// TwinCAT 3 PLC project PLC
// ProgramVersion: 3.1.4022.3
// libraries:
//   Tc2_EtherCAT, * (Beckhoff Automation GmbH)
//   Tc2_Math, * (Beckhoff Automation GmbH)
//   Tc2_Standard, * (Beckhoff Automation GmbH)
//   Tc2_System, * (Beckhoff Automation GmbH)
//   Tc2_TcpIp, * (Beckhoff Automation GmbH)
//   Tc2_Utilities, * (Beckhoff Automation GmbH)
//   Tc3_JsonXml, * (Beckhoff Automation GmbH)
//   Tc3_Module, * (Beckhoff Automation GmbH)
//   Tc3_System_DK, * (Beckhoff - DK)
// project tree:
//   DAQ/FromLib/Influxdb/Reader/ E_InfluxReaderState.TcDUT, FB_InfluxReader.TcPOU
//   DAQ/FromLib/Influxdb/Sender/ FB_InfluxDataCollector.TcPOU, FB_InfluxDataSender.TcPOU
//   DAQ/FromLib/Influxdb/Utils/ ST_InfluxBuffer.TcDUT
//   DAQ/FromLib/StringBuilder/ FB_StringBuilder.TcPOU
//   DAQ/FromLib/TcpIp Connection/ E_TcpState.TcDUT, FB_TcpConnection.TcPOU
//   DAQ/ InfluxAddData_1000Hz.TcPOU, InfluxAddData_100Hz.TcPOU, InfluxAddData_10Hz.TcPOU, InfluxAddData_1Hz.TcPOU, P_InfluxDatabaseWriter.TcPOU, P_InfluxDataCollector.TcPOU
//   DAQ/InfluxReader/ExtractValuesFromInflux/ fcnExtractInfluxData.TcPOU, ST_NumberInString.TcDUT
//   DAQ/InfluxReader/ FB_Flender_DamageReader.TcPOU, P_FlenderGetDamage.TcPOU
//   / DAQ_Collector.TcTTO, DAQ_Writer.TcTTO, MAIN.TcPOU, PlcTask.TcTTO
//   GVLs/ Communication.TcGVL, PersistentVariables.TcGVL
//   HMI/ ST_FROM_HMI.TcDUT, ST_GUI_HMI.TcDUT, ST_HOUR_COUNTERS.TcDUT, ST_PARAMETERS_HMI.TcDUT, ST_TO_HMI.TcDUT
//   Interfaces/JetsonTx2/ ST_JetsonTx2.TcDUT
//   Interfaces/Sick/ ST_SICK.TcDUT
//   Main/Enumerators/ E_EmulatedState.TcDUT
//   Main/Programs/ P_UpdateDAQ.TcPOU, P_UpdateHmi.TcPOU
//   Main/Structures/GPS/ ST_GPS.TcDUT, ST_GPS_CALCULATIONS.TcDUT, ST_GPS_INPUTS.TcDUT, ST_GPS_OUTPUTS.TcDUT
//   Main/Structures/ ST_DATA.TcDUT, ST_PlcTiming.TcDUT
// real-time tasks:
//   TASK PlcTask: cycle T#1ms, priority 20, ADS port 350
//   TASK DAQ_Collector: cycle T#10ms, priority 3, ADS port 351
//   TASK DAQ_Writer: cycle T#100000us, priority 2, ADS port 352

CONFIGURATION PLC
    RESOURCE PLC ON TwinCAT3
        TASK DAQ_Collector(INTERVAL := T#10ms, PRIORITY := 3);
        TASK DAQ_Writer(INTERVAL := T#100000us, PRIORITY := 2);
        TASK PlcTask(INTERVAL := T#1ms, PRIORITY := 20);
        PROGRAM P_InfluxDataCollector WITH DAQ_Collector : P_InfluxDataCollector;
        PROGRAM P_InfluxDatabaseWriter WITH DAQ_Writer : P_InfluxDatabaseWriter;
        PROGRAM MAIN WITH PlcTask : MAIN;
    END_RESOURCE
END_CONFIGURATION

// ---- DAQ/FromLib/Influxdb/Reader/E_InfluxReaderState.TcDUT
{attribute 'qualified_only'}
{attribute 'strict'}
TYPE E_InfluxReaderState :
(
	Idle := 0,
	Connecting,
	Query,
	ConvertingNumbers, 
	Disconnecting
) DINT;
END_TYPE

// ---- DAQ/FromLib/Influxdb/Utils/ST_InfluxBuffer.TcDUT
TYPE ST_InfluxBuffer :
STRUCT
	Initialized : BOOL;
	ReadyToSend	: BOOL;
	Data 		: FB_STRINGBUILDER; 
END_STRUCT
END_TYPE

// ---- DAQ/FromLib/TcpIp Connection/E_TcpState.TcDUT
{attribute 'qualified_only'}
{attribute 'strict'}
TYPE E_TcpState :
(
	None := 0,
	Disconnecting,
	Disconnected,
	Connecting,	
	Connected,
	Sending,
	SendingByReference,
	Waiting,
	Receiving,
	Received
) DINT;
END_TYPE

// ---- DAQ/InfluxReader/ExtractValuesFromInflux/ST_NumberInString.TcDUT
TYPE ST_NumberInString :
STRUCT
	StartIndex : DINT;
	EndIndex	: DINT; 
	Length		: DINT;
	Txt			: T_MAXSTRING;
	Value		: LREAL; 	
END_STRUCT
END_TYPE

// ---- HMI/ST_FROM_HMI.TcDUT
TYPE ST_FROM_HMI :
STRUCT
END_STRUCT
END_TYPE

// ---- HMI/ST_GUI_HMI.TcDUT
TYPE ST_GUI_HMI :
STRUCT
END_STRUCT
END_TYPE

// ---- HMI/ST_HOUR_COUNTERS.TcDUT
TYPE ST_HOUR_COUNTERS :
STRUCT
	
	TotalHours		: LTIME;
	
	WorkingHours	: LTIME;
END_STRUCT
END_TYPE

// ---- HMI/ST_PARAMETERS_HMI.TcDUT
TYPE ST_PARAMETERS_HMI :
STRUCT
END_STRUCT
END_TYPE

// ---- HMI/ST_TO_HMI.TcDUT
TYPE ST_TO_HMI :
STRUCT
	Data		: ST_DATA;
END_STRUCT
END_TYPE

// ---- Interfaces/JetsonTx2/ST_JetsonTx2.TcDUT
TYPE ST_JetsonTx2 :
STRUCT
END_STRUCT
END_TYPE

// ---- Interfaces/Sick/ST_SICK.TcDUT
TYPE ST_SICK :
STRUCT
END_STRUCT
END_TYPE

// ---- Main/Enumerators/E_EmulatedState.TcDUT
TYPE E_EmulatedState :
(
	StaticData := 0,
	SimulinkPlant,
	VirtualPlant,
	PhysicalPlant	
) DINT;
END_TYPE

// ---- Main/Structures/GPS/ST_GPS.TcDUT
TYPE ST_GPS :
STRUCT
	Inputs			: ST_GPS_INPUTS;
	Outputs			: ST_GPS_OUTPUTS;
	Calculations	: ST_GPS_CALCULATIONS;
END_STRUCT
END_TYPE

// ---- Main/Structures/GPS/ST_GPS_CALCULATIONS.TcDUT
TYPE ST_GPS_CALCULATIONS :
STRUCT
END_STRUCT
END_TYPE

// ---- Main/Structures/GPS/ST_GPS_INPUTS.TcDUT
TYPE ST_GPS_INPUTS :
STRUCT
	x			: LREAL;
END_STRUCT
END_TYPE

// ---- Main/Structures/GPS/ST_GPS_OUTPUTS.TcDUT
TYPE ST_GPS_OUTPUTS :
STRUCT
END_STRUCT
END_TYPE

// ---- Main/Structures/ST_DATA.TcDUT
TYPE ST_DATA :
STRUCT
	Timing				: ST_PlcTiming;
	JetsonTx2			: ST_JetsonTx2;
	Sick				: ST_SICK;
	Gps					: ST_Gps;
END_STRUCT
END_TYPE

// ---- Main/Structures/ST_PlcTiming.TcDUT
TYPE ST_PlcTiming :
STRUCT
	TimeStamp 		: T_FILETIME;  	(* Current Windows timestamp *)
	UnixTimeStamp 	: ULINT; 		(* Number of 100 ns since 1.1.1970 *)
	SpanTime		: LTIME;		(* PLC RunTime*)

	ScanTime		: LTIME; 		(* TIME: PLC Scantime *)
	ScanTime_s		: LREAL; 		(* LREAL: PLC Scantime in seconds *)
	ScanTime_ms		: LREAL	:= ScanTime_s * 1E3;		(* LREAL: PLC Scantime in milli seconds *)
	
	Tick			: UDINT := 0; 	(* Current PLC tick count *)
	Toggle			: BOOL; 		(* BOOL: Toggle Each Scan *)
	Toggle1Hz		: BOOL; 		(* BOOL: Toggle at 1 Hz: 1000 ms *)
	Toggle100Hz		: BOOL; 		(* BOOL: Toggle at 100 Hz: 10 ms*)
END_STRUCT
END_TYPE

// ---- GVLs/Communication.TcGVL
{attribute 'qualified_only'}
VAR_GLOBAL
	ToHmi				: ST_TO_HMI;
	
	FromHmi				: ST_FROM_HMI;
	
	Parameters 			: ST_PARAMETERS_HMI;

	Gui					: ST_GUI_HMI; 
	
	HourCounters		: ST_HOUR_COUNTERS;
	
	// Temp
	MyBoolVariable		: BOOL;
END_VAR

// ---- GVLs/PersistentVariables.TcGVL
{attribute 'qualified_only'}
VAR_GLOBAL
	HourCounters		: ST_HOUR_COUNTERS;
END_VAR

// ---- DAQ/P_InfluxDataCollector.TcPOU
PROGRAM P_InfluxDataCollector
VAR 
	Data : REFERENCE TO ST_DATA := P_UpdateDAQ.DataDaq;  
	Tick : LREAL; 
	ActualBufferTime : TIME; 
	
	InfluxData : FB_InfluxDataCollector; 

	Timer1Hz 	: TON; 
	Timer10Hz 	: TON; 
	Timer100Hz 	: TON; 	

END_VAR

Tick := Tick + 1;
RunTimers(); 

// ========= Initialize Data
	InfluxData.Initialize( 	HostName 		:= 'MachinePLC',			// <<---- 	Change to Descriptive MachinePLC name, eg: MachinePLC_TLU 
							Database 		:= 'RD',			// <<---- 	Change to Database name. Needs to be setup beforehand.
							Measurement 	:= 'CKD_Test');	// <<---- 	Measurentname in database. Eg: LORCHALT
// ========= Add Data tags.
// These are written to each "point" i.e. for each ms.
// Add eg: Current State of TestBench - for easy search later on
															
	//Data.AddTag('State','Default');						

// ========= Add Actual Data

	InfluxData.AddLreal('Tick', Tick);

// ======== 1 Hz Data
	IF Time_1Hz THEN
		InfluxData.AddLreal('Test1Hz', 1);	
	
		InfluxAddData_1Hz(		Data 			:= Data,
								DataCollector 	:=  InfluxData); 	
						
	END_IF
	
// ======== 10 Hz Data
	IF Time_10Hz THEN
		InfluxData.AddLreal('Test10Hz', 10);
	
		InfluxAddData_10Hz(	Data 			:= Data,
								DataCollector 	:=  InfluxData); 		
		
	END_IF

// ======== 100 Hz Data
	IF Time_100Hz THEN
		InfluxData.AddLreal('Test100Hz', 100);
	
		InfluxAddData_100Hz(	Data 			:= Data,
								DataCollector 	:=  InfluxData); 

		InfluxAddData_1000Hz(	Data 			:= Data,
								DataCollector 	:=  InfluxData); 
	
								
	END_IF


// =========== Add TimeStamp and start new "point"
InfluxData.AddTimeStamp(ActualBufferTime => ActualBufferTime); 















ResetTimersIfDone();

METHOD ResetTimersIfDone : BOOL
IF Timer1Hz.Q THEN
	Timer1Hz(IN := FALSE); 
	Timer1Hz(IN := TRUE); 

END_IF
IF Timer10Hz.Q THEN
	Timer10Hz(IN := FALSE); 
	Timer10Hz(IN := TRUE); 
	

END_IF
IF Timer100Hz.Q THEN
	Timer100Hz(IN := FALSE); 
	Timer100Hz(IN := TRUE); 
	
END_IF
END_METHOD

METHOD RunTimers : BOOL
Timer1Hz(	IN := TRUE, PT := T#1S		); 
Timer10Hz(	IN := TRUE, PT := T#100MS	); 
Timer100Hz(	IN := TRUE, PT := T#10MS	);
END_METHOD

PROPERTY Time_100Hz : BOOL
GET
Time_100Hz := Timer100Hz.Q;
END_GET
END_PROPERTY

PROPERTY Time_10Hz : BOOL
GET
Time_10Hz := Timer10Hz.Q;
END_GET
END_PROPERTY

PROPERTY Time_1Hz : BOOL
GET
Time_1Hz := Timer1Hz.Q;
END_GET
END_PROPERTY

END_PROGRAM

// ---- Main/Programs/P_UpdateDAQ.TcPOU
PROGRAM P_UpdateDAQ
VAR_IN_OUT
	Data	: ST_DATA;
END_VAR
VAR
	DataDaq : ST_DATA;
END_VAR

DataDaq := Data;

END_PROGRAM

// ---- DAQ/FromLib/Influxdb/Sender/FB_InfluxDataCollector.TcPOU
FUNCTION_BLOCK FB_InfluxDataCollector
VAR
//Writer
	_NameValuePairs			: UDINT; 
	_PointsAdded			: UDINT; 
	
// Misc
	_fbGetSystemTime		: GetSystemTime;
	_bufferTime				: TIME; 
	_fbTimer				: TON; 
END_VAR
VAR
	BufferInUse		: DINT := 1; 
	Buffer1			: ST_InfluxBuffer;
	Buffer2			: ST_InfluxBuffer;
END_VAR
VAR
	iContentLengthIndex : UDINT; 
	iContentLengthBegin : UDINT;
	iContentLengthEnd	: UDINT;
	iContentLength		: UDINT; 
	strContentLength	: T_MAXSTRING; 
END_VAR

METHOD AddBareString : BOOL
VAR_INPUT
	input : T_MaxString; 
END_VAR
DataString.Append(input);
END_METHOD

METHOD PUBLIC AddBool : BOOL
VAR_INPUT
	Name 	: T_MaxString;
	Value 	: BOOL; 
END_VAR
AddName(Name);
IF Value THEN
	DataString.Append('1');
ELSE
	DataString.Append('0');
END_IF
END_METHOD

METHOD PUBLIC AddData : BOOL
VAR_INPUT
	Name 	: T_MaxString;
	Value 	: T_MaxString; 
END_VAR
AddName(Name);
DataString.Append(Value);


_NameValuePairs := _NameValuePairs + 1;
END_METHOD

METHOD AddLreal : BOOL
VAR_INPUT
	Name 	: T_MaxString;
	Value 	: LREAL; 
END_VAR
VAR_INST
	json	: FB_JsonSaxWriter; 
END_VAR
AddName(Name);

json.ResetDocument(); 
json.AddLreal(Value); 
DataString.Append(json.GetDocument());
END_METHOD

METHOD PRIVATE AddName : BOOL
VAR_INPUT
	Name 	: T_MaxString;
END_VAR
IF _NameValuePairs = 0 THEN
	DataString.Append(' ');
ELSE
	DataString.Append(',');
END_IF
DataString.Append(Name);
DataString.Append('=');

_NameValuePairs := _NameValuePairs + 1;
END_METHOD

METHOD AddTag : BOOL
VAR_INPUT
	Key		: T_MAXSTRING;
	Value	: T_MAXSTRING; 
END_VAR
Datastring.Append(',');
Datastring.Append(Key);
DataString.Append('=');
DataString.Append(Value);
END_METHOD

METHOD AddTimeStamp : BOOL; 

VAR
	b : BOOL; 
	SizeLimit : UDINT := 10000000; //10 MB
END_VAR
VAR_OUTPUT
	ActualBufferTime : TIME; 
END_VAR
VAR_INST
	_actualBufferTime : TIME; 
END_VAR
_PointsAdded := _PointsAdded + 1;

DataString.Append(' ');
DataString.Append(ULINT_TO_STRING(CurrentTimeStamp));
DataString.Append('$N');

_fbTimer(	IN := TRUE,
			PT := _bufferTime);
			
IF _fbTimer.Q OR BufferUsed >= 0.9 OR DataString.Length > SizeLimit THEN
	_actualBufferTime := _fbTimer.ET;

	// ======= Add HTTP Content Length
	
		iContentLengthEnd := DataString.Length; 
		
		// Calcualte ContentLength 
		iContentLength := iContentLengthEnd - iContentLengthBegin; 
		strContentLength := TO_STRING(iContentLength); 
		
		// Add content Length to HTTP Header
		memcpy(DataString.StringPointer + iContentLengthIndex, ADR(strContentLength), LEN(strContentLength));


	SetBufferAsReady();
	SwitchBuffer(); 
	Reset(); 
	SetBufferAsNotReady();
	
	
	
	
END_IF

ActualBufferTime := _actualBufferTime;
END_METHOD

PROPERTY BufferOverflow : BOOL
GET
BufferOverflow := DataString.Length = DataString.BufferSize;
END_GET
END_PROPERTY

PROPERTY BufferUsed : LREAL
GET
BufferUsed := UDINT_TO_LREAL(DataString.Length) / UDINT_TO_LREAL(DataString.BufferSize);
END_GET
END_PROPERTY

PROPERTY PROTECTED CurrentTimeStamp : ULINT;
GET
VAR
	normTime	: T_FILETIME;

	dcTime	: T_DCTIME64; 	

	timeLoDW				: ULINT;
	timeHiDW				: ULINT;
	ulTime					: ULINT;
	unixTimeFileTimeDiff	: ULINT;

	
END_VAR
(****************************************************************************************************************

In TwinCAT we get accure timestamp  via GetSystemTime() function block, but it returns so called "filetime"
	filemtime is count of "100 nanoseconds" since 1.1.1601.
	
InfluxDb uses Unix time stamp with accuracy of 1ns. 
	Unix time stamp is seconds since 1.1.1970. 

1.1.1970 - 1.1.1601 in "100 nanoseconds" is 116444736000000000	
*******************************************************************************************************************)

unixTimeFileTimeDiff := 116444736000000000; 
_fbGetSystemTime();
timeHiDW 	:= _fbGetSystemTime.timeHiDW;
timeLoDW 	:= _fbGetSystemTime.timeLoDW; 


normTime := DCTIME64_TO_FILETIME(F_GETCURDCTASKTIME64()); 

normTime.dwHighDateTime := normTime.dwHighDateTime;
normTime.dwLowDateTime := normTime.dwLowDateTime;


ulTime 	:= timeHiDW * 16#FFFFFFFF + timeLoDW; 	// "100 nanoseconds" since 1.1.1601.

//ulTime 	:= normTime.dwHighDateTime * 16#FFFFFFFF + normTime.dwLowDateTime; 	// "100 nanoseconds" since 1.1.1601.

ulTime 	:= ulTime - unixTimeFileTimeDiff;		// "100 nanoseconds" since 1.1.1970.
CurrentTimeStamp 	:= ulTime * 100;						// nanoseconds since 1.1.1970.
END_GET
END_PROPERTY

PROPERTY DataLength : UDINT
GET
DataLength := DataString.Length;
END_GET
END_PROPERTY

PROPERTY DataString : REFERENCE TO FB_STRINGBUILDER
GET
DataString REF= GetData(BufferInUse);
END_GET
END_PROPERTY

METHOD GetData : REFERENCE TO FB_STRINGBUILDER
VAR_INPUT
	BufferNumber : DINT; 
END_VAR

IF BufferNumber = 1 THEN
	GetData REF= Buffer1.Data;
ELSIF BufferNumber = 2 THEN
	GetDAta REF= Buffer2.Data; 
END_IF
END_METHOD

PROPERTY HttpRequest : T_MAXSTRING
GET
HttpRequest := DataString.ToString;
END_GET
END_PROPERTY

METHOD Initialize : BOOL
VAR_INPUT
	HostName 		: T_MAXSTRING;
	Database 		: T_MAXSTRING;  
	Measurement 	: T_MAXSTRING; 
END_VAR
VAR
	MaxBufferTime : TIME := T#2s; 
END_VAR
IF DataString.Length = 0 THEN
	// ============ Build HTTP Header
	DataString.Append('POST /write?db=');
	DataString.Append(Database);
	DataString.AppendLine(' HTTP/1.1');
	
	DataString.Append('Host: ');
	DataString.AppendLine(HostName);
	DataString.AppendLine('User-Agent: TwinCAT HttpClient');
	DataString.AppendLine('Content-Type: application/x-www-form-urlencoded');
	
	DataString.Append('Content-Length: ');
	iContentLengthIndex := DataString.Length; 
	
	DataString.Append('                    '); // Add 10 spaces for adding ContentLength later;
	DataString.AppendLine('');
	DataString.AppendLine(''); 	// <<--- End of HTTP Header
	
	iContentLengthBegin := DataString.Length; 
END_IF

	
// ========== Add host to influx measurement
SetupCollection(Measurement, HostName, MaxBufferTime);
END_METHOD

METHOD IsReadyToSend : BOOL
VAR_INPUT
	BufferNumber : DINT; 
END_VAR
IF BufferNumber = 1 THEN
	IsReadyToSend := Buffer1.ReadyToSend; 
ELSIF BufferNumber = 2 THEN
	IsReadyToSend := Buffer2.ReadyToSend;  
END_IF
END_METHOD

PROPERTY PointsAdded : UDINT
GET
PointsAdded := _PointsAdded;
END_GET
END_PROPERTY

PROPERTY ReadyToSend : BOOL
GET
ReadyToSend := _fbTimer.Q;
END_GET
END_PROPERTY

METHOD Reset : BOOL
VAR_INPUT
END_VAR
_fbTimer(IN := FALSE);
DataString.Clear();
_PointsAdded := 0;
END_METHOD

METHOD PRIVATE SetBufferAsNotReady : BOOL

// ========== Current
IF BufferInUse = 1 THEN
	Buffer1.ReadyToSend := FALSE;
ELSIF BufferInUse = 2 THEN
	Buffer2.ReadyToSend := FALSE;
END_IF
END_METHOD

METHOD PRIVATE SetBufferAsReady : BOOL

// ========== Current
IF BufferInUse = 1 THEN
	Buffer1.ReadyToSend := TRUE;
ELSIF BufferInUse = 2 THEN
	Buffer2.ReadyToSend := TRUE;
END_IF
END_METHOD

METHOD SetupCollection : BOOL; 
VAR_INPUT
	Measurement				: T_MaxString;
	ComputerName			: T_MaxString;
	BufferTime				: TIME; 
END_VAR
DataString.Append(Measurement);

AddTag('Source',ComputerName);


_bufferTime := BufferTime; 


_NameValuePairs := 0;
END_METHOD

METHOD PRIVATE SwitchBuffer : BOOL
IF BufferInUse = 1 THEN
	BufferInUse := 2; 
ELSE
	BufferInUSe := 1; 
END_IF
END_METHOD

PROPERTY TagsAdded : UDINT
GET
TagsAdded := _NameValuePairs;
END_GET
END_PROPERTY

PROPERTY TimeElapsed : TIME
GET
TimeElapsed := _fbTimer.ET;
END_GET
END_PROPERTY

PROPERTY TimeRemaining : TIME
GET
TimeRemaining := _bufferTime - TimeElapsed;
END_GET
END_PROPERTY

PROPERTY ToString : T_MAXSTRING
GET
ToString := DataString.ToString;
END_GET
END_PROPERTY

END_FUNCTION_BLOCK

// ---- DAQ/FromLib/StringBuilder/FB_StringBuilder.TcPOU
FUNCTION_BLOCK FB_StringBuilder

VAR
	{attribute 'hide'}
	_dataBuffer		: ARRAY[0..MaxBufferSize] OF BYTE;  // Buffer for storing of all text
	_dataBufferAdd 	: POINTER TO BYTE; // Databuffer start adress
	_currentLength 	: UDINT; // Current length of string in databuffer. 
END_VAR

VAR CONSTANT
	MaxBufferSize : UDINT := 49999999; // max 50MB buffer 	
END_VAR

METHOD Append : BOOL
VAR_INPUT
	InputString : T_MaxString;
END_VAR
VAR
	StringLength: UDINT;
END_VAR

StringLength := DINT_TO_UDINT(LEN(InputString));
Append := THIS^.AppendGeneric(ADR(InputString),StringLength);
END_METHOD

METHOD AppendGeneric : BOOL
VAR_INPUT
	AddressPointer : POINTER TO BYTE; // Pointer to data
	DataLength : UDINT; 
END_VAR
IF _dataBufferAdd = 0 THEN
	_dataBufferAdd := ADR(_dataBuffer);
END_IF

IF _currentLength + DataLength < MaxBufferSize AND DataLength > 0 THEN
	MEMCPY(_dataBufferAdd + _currentLength, AddressPointer, DataLength);
	_currentLength := _currentLength + DataLength;
	AppendGeneric := TRUE;
ELSE
	AppendGeneric := FALSE;
END_IF
END_METHOD

METHOD AppendLine : BOOL
VAR_INPUT
	InputString : T_MaxString;
END_VAR
THIS^.Append(InputString);
THIS^.Append('$R$N');
END_METHOD

PROPERTY BufferSize : UDINT
GET
BufferSize := MaxBufferSize;
END_GET
END_PROPERTY

METHOD Clear : BOOL
VAR_INPUT
END_VAR
_currentLength := 0;
END_METHOD

METHOD GetIndexOf : DINT
VAR_INPUT
	SearchString	: T_MAXSTRING; 
	StartIndex		: UDINT;
END_VAR
VAR
	searchStringLength : UDINT;
	
	iStringIndex	: UDINT;

	
	matchFound 	: BOOL;

	

 
END_VAR



searchStringLength := TO_UDINT(LEN(SearchString));

IF StartIndex < 0 THEN
	StartIndex := 0;
END_IF

matchFound := FALSE; 
IF (searchStringLength <= THIS^.Length) AND (StartIndex <  THIS^.Length-searchStringLength) THEN
	FOR iStringIndex := StartIndex TO (THIS^.Length-searchStringLength) DO
		// Loop through current string.
	
		
		// Search for string
		
		matchFound := memcmp(	pBuf1 	:= THIS^.StringPointer + iStringIndex,
								pBuf2 	:= ADR(SearchString),
								n		:= searchStringLength) = 0;  
	
	
		IF matchFound THEN
			EXIT;
		END_IF
	END_FOR
END_IF
IF matchFound THEN
	GetIndexOf := TO_DINT(iStringIndex); 
ELSE
	GetIndexOf := -1;
END_IF
END_METHOD

METHOD Initialize : BOOL
IF _dataBufferAdd = 0 THEN
	_dataBufferAdd := ADR(_dataBuffer);
END_IF
END_METHOD

PROPERTY Length : UDINT
GET
Length := _currentLength;
END_GET
SET
_currentLength := Length;
END_SET
END_PROPERTY

PROPERTY StringPointer : POINTER TO BYTE
GET
StringPointer := _dataBufferAdd;
END_GET
END_PROPERTY

PROPERTY ToString : STRING(255)
GET
VAR_INST
	s255String : STRING(255);
	length : UDINT;
END_VAR
s255String := '';
length := MIN(_currentLength, DINT_TO_UDINT(SIZEOF(s255String)));
MEMCPY(ADR(s255String), _dataBufferAdd, length);
ToString := s255String;
END_GET
END_PROPERTY

PROPERTY ToStringEnding : STRING(255)
GET
VAR_INST
	s255String : STRING(255);
	length : UDINT;
END_VAR
s255String := '';
length := 255;
IF _currentLength > 255 THEN
	MEMCPY(ADR(s255String), _dataBufferAdd+_currentLength-length, length);
ELSE
	s255String := 'Length less than 255'; 
END_IF
ToStringEnding := s255String;
END_GET
END_PROPERTY

END_FUNCTION_BLOCK

// ---- DAQ/InfluxAddData_1Hz.TcPOU
FUNCTION InfluxAddData_1Hz : BOOL
VAR_IN_OUT
	Data			: ST_DATA;
	DataCollector	: FB_InfluxDataCollector;
END_VAR

// Damage counter values
DataCollector.AddLreal('Test2',		Data.Gps.Inputs.x);

END_FUNCTION

// ---- DAQ/InfluxAddData_10Hz.TcPOU
FUNCTION InfluxAddData_10Hz : BOOL
VAR_IN_OUT
	Data			: ST_DATA;
	DataCollector	: FB_InfluxDataCollector;
END_VAR

// =================== Example:
	DataCollector.AddLreal(	'Test',                      Data.Gps.Inputs.x);

END_FUNCTION

// ---- DAQ/InfluxAddData_100Hz.TcPOU
FUNCTION InfluxAddData_100Hz : BOOL
VAR_IN_OUT
	Data			: ST_DATA;
	DataCollector	: FB_InfluxDataCollector;
END_VAR

// =================== Test
	DataCollector.Addlreal(	'Test64',                                    Data.Gps.Inputs.x);

END_FUNCTION

// ---- DAQ/InfluxAddData_1000Hz.TcPOU
FUNCTION InfluxAddData_1000Hz : BOOL
VAR_IN_OUT
	Data	: ST_DATA;
	DataCollector	: FB_InfluxDataCollector;
END_VAR

// =================== Test
	DataCollector.AddLreal(	'Test3',                                         Data.Gps.Inputs.x);

END_FUNCTION

// ---- DAQ/P_InfluxDatabaseWriter.TcPOU
PROGRAM P_InfluxDatabaseWriter
VAR
	Data : REFERENCE TO FB_InfluxDataCollector := P_InfluxDataCollector.InfluxData; 	

	Sender : FB_InfluxDataSender; 
	
	WriteSucces : BOOL; 
END_VAR

(* This Sender Program Should be run at 10ms ScanTime in seperate task (can be same CPU) from DataCollector *)

IF Main.EmulatedState = E_EmulatedState.PhysicalPlant THEN
	Sender(	Data				:= Data,
			Ip					:= '10.10.0.122',
			Port				:= 8086,
			GlobalWriteSucces 	=> WriteSucces); 
ELSIF Main.EmulatedState = E_EmulatedState.VirtualPlant THEN
	Sender(	Data				:= Data,
			Ip					:= '127.0.0.1',
			Port				:= 8086,
			GlobalWriteSucces 	=> WriteSucces); 	

END_IF



// =============== Read Values from Influxdb

END_PROGRAM

// ---- DAQ/FromLib/Influxdb/Sender/FB_InfluxDataSender.TcPOU
FUNCTION_BLOCK FB_InfluxDataSender
VAR_INPUT
	Data 		: REFERENCE TO FB_InfluxDataCollector; 
	Ip			: T_IPv4Addr := '127.0.0.1';	(* IP Adress for TCP/IP Server *)
	Port 		: UDINT := 8086; 				(* Port To Connect to *)
END_VAR
VAR_OUTPUT
	GlobalWriteSucces	: BOOL;
END_VAR
VAR CONSTANT
	BufferLength : DINT := 2; 
END_VAR
VAR
	ResetConnection : BOOL; 
END_VAR

VAR
	i : DINT; 
	iTest : UDINT; 	
	currentBytes : UDINT; 

	tcp 			: ARRAY[1..BufferLength] OF FB_TcpConnection; 
	CurrentState 	: ARRAY[1..BufferLength] OF E_TcpState; 
	Connected 		: ARRAY[1..BufferLength] OF BOOL; 
	
	RisingEdge 		: ARRAY[1..BufferLength] OF R_TRIG; 
	FallingEdge		: ARRAY[1..BufferLength] OF F_TRIG; 	
	
	SendCounter 	: ARRAY[1..BufferLength] OF UDINT;
	
	WriteSucces 	: ARRAY[1..BufferLength] OF BOOL; 
END_VAR
VAR
	ShiftCounter : CTU;
	ShiftCounted : UDINT; 
END_VAR

iTest := iTest + 1;  

IF __ISVALIDREF(Data) THEN
	GlobalWriteSucces := TRUE;
	FOR i := 1 TO BufferLength DO
		
		
		
		IF ResetConnection THEN
			tcp[i].Disconnect(); 
		END_IF	
	
		
		tcp[i](	Ip 					:= Ip,//'192.168.1.209',
				Port				:= 8086,
				ReplyReadInterval 	:= T#100MS); 
				
		CurrentState[i] := tcp[i].State; 		
		Connected[i] := tcp[i].Connected; 		
	
		RisingEdge[i](CLK := Data.IsReadyToSend(i));
		FallingEdge[i](CLK := Data.IsReadyToSend(i));
		
		IF RisingEdge[i].Q THEN
			currentBytes := Data.GetData(i).Length;
			tcp[i].Send(Data.GetData(i).StringPointer, Data.GetData(i).Length);
			SendCounter[i] := SendCounter[i] + 1;  	
		END_IF
		IF FallingEdge[i].Q THEN
			tcp[i].Connect();		
		END_IF
		
		
		
		//IF tcp[i].
		
		IF CurrentState[i] < E_TcpState.Connected THEN
			WriteSucces[i] := FALSE; 
		ELSIF CurrentState[i] = E_TcpState.Received THEN
			WriteSucces[i] := (memcmp(tcp[i].Response.StringPointer,ADR('HTTP/1.1 204 No Content'),20) = 0) 
								AND tcp[i].ResponseReceived;
		END_IF
		
	END_FOR
	
	GlobalWriteSucces := WriteSucces[1] AND WriteSucces[2];
	ShiftCounter(CU := GlobalWriteSucces, PV := 200, CV => ShiftCounted);
ELSE
	GlobalWriteSucces := FALSE; 
END_IF

END_FUNCTION_BLOCK

// ---- DAQ/FromLib/TcpIp Connection/FB_TcpConnection.TcPOU
(* Generic TcpIp Connection  *) 
FUNCTION_BLOCK FB_TcpConnection
VAR_INPUT
	Ip					: T_IPv4Addr; (* IP Adress for TCP/IP Server *)
	Port 				: UDINT; (* Port To Connect to *)
	ReplyReadInterval 	: TIME := T#100MS; (* Time for allowing server to start responding [T#100MS]*)
END_VAR
VAR_OUTPUT
	_response 	: FB_StringBuilder;
END_VAR

VAR
	_requestAdr		: POINTER TO BYTE;
	_requestLength	: UDINT; 	
	
	_responseBuilder : FB_StringBuilder; 
	
	_responseString	: T_MAXSTRING; 
	_responseReceived	: BOOL; 
	_handle		: T_HSOCKET; 
	
	// ======== Current Connection
	_connect	: BOOL; 
	_connected	: BOOL; 

	_lastState		: E_TcpState; 
	_currentState	: E_TcpState :=  E_TcpState.Disconnected;

	// ======== ErrorString
	_errorID				: UDINT; 
	_errorMsg				: T_MAXSTRING; 

	// ======== Internal Stuff
	_idleTime	: TIME;
	_timeInState : TIME; 
	_stateCycles : UDINT;
	_firstTimeInState : BOOL; 
	
	// ======== Optional stuff
	_AmsNetId	: T_AmsNetID := ''; // Local host
	_Timeout	: TIME := T#45S; 
	
	
END_VAR

(*
Eventlog:
18-08-2018 - JHH - Created



*)


// ========== Initialize Buffers
_response.Initialize();

UpdateMetrics(	CurrentState 	:= _CurrentState,
				IdleTime		=> _IdleTime,
				TimeInState		=> _timeInState,
				CyclesInState 	=> _stateCycles, 
				FirstTimeInState => _firstTimeInState); 

_lastState := _currentState;
CASE _currentState OF
	// ============== Connect
		E_TcpState.Connecting:
			state_Connecting(		Handle			:= _handle,
									CurrentState	:= _currentState,
									Ip				:= Ip,
									Port			:= Port);	
		
		E_TcpState.Connected:
			state_Connected(		Connected		:= _connected); 
			
	// ============== Send/Receive	
		E_TcpState.Sending:

			state_Sending(			RequestAdr		:= _requestAdr,
									RequestLength	:= _requestLength,
									ResponseBuilder	:= _responseBuilder,
									CurrentState	:= _currentState,
									Handle			:= _handle);
									
								
									
		E_TcpState.Waiting:
			state_Waiting(			CurrentState	:= _currentState,
									WaitTime		:= ReplyReadInterval);
		
		E_TcpState.Receiving:

			state_Receiving(		ResponseBuilder := _responseBuilder,
									ActualResponse		:= _response,
									CurrentState	:= _currentState,
									Handle			:= _handle); 

						
		E_TcpState.Received:
			state_Received(			CurrentState	:= _currentState); 
									
	// ============== DisConnect							
		E_TcpState.Disconnecting:
			state_Disconnecting(	Handle			:= _handle,
									CurrentState	:= _currentState);	
	
		E_TcpState.Disconnected:
			state_Disconnected(		Connected		:= _connected);	
	
END_CASE

 
//_requestString := _request.ToString;


_errorMsg := ErrorIdToString(	ErrorID 		:= _errorID);

PROPERTY Busy : BOOL
GET
Busy := 	_currentState = E_TcpState.Receiving 
		OR	_currentState = E_TcpState.Sending
		OR	_currentState = E_TcpState.Waiting;
END_GET
END_PROPERTY

METHOD Connect : BOOL
IF _currentState = E_TcpState.Disconnected THEN
	_currentState := E_TcpState.Connecting; 
END_IF
END_METHOD

PROPERTY Connected : BOOL
GET
Connected := _connected;
END_GET
END_PROPERTY

METHOD Disconnect : BOOL
VAR_INPUT
END_VAR
_currentState := E_TcpState.Disconnecting;
END_METHOD

METHOD PRIVATE ErrorIdToString : T_MAXSTRING
VAR_INPUT
	ErrorID	: UDINT; 
END_VAR
CASE ErrorID OF
	0: 	
		ErrorIdToString := 'No Error';
	32769:
		ErrorIdToString := 'TCP/IP Connection Server: No new sockets can be created';
	32770:
		ErrorIdToString := 'TCP/IP Connection Server: Socket handle is invalid';
	32771:
		ErrorIdToString := 'TCP/IP Connection Server: TcpIp port listener already exists';
	32772:
		ErrorIdToString := 'TCP/IP Connection Server: Client socket is no longer connected with the server.';
	32773:
		ErrorIdToString := 'TCP/IP Connection Server: Error was registered in the listener socket.';
		
	2147952453:
		ErrorIdToString	:= 'Win32 Socket: An established connection was aborted BY the software in your host machine.';
		
	2147952454:
		ErrorIdToString	:= 'Win32 Socket: An existing connection was forcibly closed by the remote host..';
	 
ELSE
	ErrorIdToString := CONCAT('Unknown Error: ',TO_STRING(ErrorID));

END_CASE
END_METHOD

PROPERTY LastErrorMsg : T_MAXSTRING
GET
LastErrorMsg := _errorMsg;
END_GET
END_PROPERTY

METHOD PRIVATE MaintainConnection : BOOL
VAR_INPUT
	ServerIp		: T_IPv4Addr;
	ServerPort 		:  UDINT; 
	Connect			: BOOL; 
END_VAR

VAR_OUTPUT
	Handle				: T_HSOCKET; 
	ConnectionState		: E_SocketConnectionState; 
	Connected			: BOOL; 
	ErrorMsg			: T_MAXSTRING; 
END_VAR

VAR_INST
	_fbConnection		: FB_ClientServerConnection; 
	

END_VAR
_fbConnection(	sSrvNetID	:= , 
				nMode		:= 0, 
				sRemoteHost	:= ServerIp, 
				nRemotePort	:= ServerPort, 
				bEnable		:= Connect, 
				tReconnect	:= T#45S, 
				bBusy		=> , 
				bError		=> , 
				nErrId		=> , 
				hSocket		=> Handle, 
				eState		=> ConnectionState);
				
Connected := ConnectionState = 	E_SocketConnectionState.eSOCKET_CONNECTED;	
ErrorMsg := ErrorIdToString(_fbConnection.nErrId);
END_METHOD

METHOD ResetError : BOOL
_errorId := 0; 
_errorMsg := ErrorIdToString(_errorId);
END_METHOD

PROPERTY Response : REFERENCE TO FB_StringBuilder
GET
Response REF= _response;
END_GET
END_PROPERTY

PROPERTY ResponseReceived : BOOL
GET
ResponseReceived := _responseReceived;
END_GET
END_PROPERTY

METHOD Send : BOOL
VAR_INPUT
	RequestAdr	: POINTER TO BYTE;
	RequestLength	: UDINT; 
END_VAR
_responseBuilder.Clear();

_requestAdr	:= RequestAdr;
_requestLength := RequestLength; 

IF _currentState = E_TcpState.Connected THEN
	_currentState := E_TcpState.Sending;
END_IF
END_METHOD

PROPERTY State : E_TcpState
GET
State := _currentState;
END_GET
END_PROPERTY

METHOD private state_Connected : BOOL
VAR_IN_OUT
	Connected		: BOOL; 
END_VAR
Connected := TRUE;
END_METHOD

METHOD PRIVATE state_Connecting : BOOL
VAR_INPUT
	Ip					: T_IPv4Addr; (* IP Adress for TCP/IP Server *)
	Port 				: UDINT; (* Port To Connect to *)
END_VAR
VAR_IN_OUT
	Handle			: T_HSOCKET;
	CurrentState	: E_TcpState;		
END_VAR
VAR_INST
	fb				: FB_SocketConnect; 
	error			: T_MAXSTRING; 
END_VAR

fb(	sSrvNetId	:= _AmsNetId, 
	sRemoteHost	:= Ip, 
	nRemotePort	:= Port, 
	bExecute	:= NOT(_firstTimeInState), 
	tTimeout	:= _Timeout, 
	bBusy		=> , 
	bError		=> , 
	nErrId		=> , 
	hSocket		=> Handle);

IF fb.bError AND NOT(_firstTimeInState) THEN
	fb(bExecute := FALSE);
	error := ErrorIdToString(fb.nErrId); 
	CurrentState := E_TcpState.Disconnecting;

ELSIF NOT(fb.bBusy) AND NOT(_firstTimeInState) THEN
	fb(bExecute := FALSE);
	CurrentState := E_TcpState.Connected;
END_IF

_errorID := fb.nErrId;
END_METHOD

METHOD PRIVATE state_Disconnected : BOOL
VAR_IN_OUT
	Connected		: BOOL; 
END_VAR
Connected := FALSE; 
_connect := FALSE;
END_METHOD

METHOD private state_Disconnecting : BOOL
VAR_IN_OUT
	Handle			: T_HSOCKET;
	CurrentState	: E_TcpState;		
END_VAR
VAR_INST
	fb				: FB_SocketClose; 
	error 			: T_MAXSTRING;
END_VAR

fb(	sSrvNetId	:= _AmsNetId, 
	hSocket		:= Handle, 
	bExecute	:= NOT(_firstTimeInState), 
	tTimeout	:= _Timeout, 
	bBusy		=> , 
	bError		=> , 
	nErrId		=> );

IF (fb.bError OR NOT(fb.bBusy)) AND NOT(_firstTimeInState) THEN
	fb(bExecute := FALSE);
	error := ErrorIdToString(fb.nErrId); 
	CurrentState := E_TcpState.Disconnected;
END_IF

_errorID := fb.nErrId;
END_METHOD

METHOD state_Received : BOOL
VAR_IN_OUT
	CurrentState	: E_TcpState; 
END_VAR
IF NOT(_firstTimeInState) THEN
	CurrentState := E_TcpState.Connected; 
	
	_responseString 	:= _response.ToString; 
	_responseReceived	:= _response.Length > 0;

END_IF
END_METHOD

METHOD private state_Receiving : BOOL
VAR_IN_OUT
	ResponseBuilder	: FB_StringBuilder; 
	ActualResponse		: FB_StringBuilder;
END_VAR
VAR_IN_OUT
	Handle			: T_HSOCKET;
	CurrentState	: E_TcpState;		
END_VAR
VAR_INST
	fb				: FB_SocketReceive; 
	ErrorID			: UDINT; 
	TxtReceived		: T_MAXSTRING; 
	error 			: T_MAXSTRING;
	buffer			: ARRAY[0..1023] OF BYTE;
	InBuffer		: UDINT; 
END_VAR

fb(
	sSrvNetId	:= _AmsNetId, 
	hSocket		:= Handle, 
	bExecute	:= NOT(_firstTimeInState),
	cbLen		:= SIZEOF(buffer), //Response.BufferSize-Response.Length, 
	pDest		:= ADR(buffer), //Response.StringPointer + Response.Length, 
	tTimeout	:= T#500h, 
	bBusy		=> , 
	bError		=> , 
	nErrId		=> ErrorID, 
	nRecBytes	=> InBuffer); //BytesReceived);

IF fb.bError AND NOT(_firstTimeInState) THEN
	fb(bExecute := FALSE);
	error := ErrorIdToString(fb.nErrId); 
	CurrentState := E_TcpState.Disconnected;

ELSIF NOT(fb.bBusy) AND NOT(_firstTimeInState) THEN
	fb(bExecute := FALSE);
	
	// ========== Transfer to Response
	ResponseBuilder.AppendGeneric(ADR(buffer), InBuffer); 
	
	
	
	
	IF InBuffer > 0 THEN
		CurrentState := E_TcpState.Waiting;	// If not all bytes received, read again in "wait" time.
	ELSE
		CurrentState := E_TcpState.Received; // If no bytes read, reading is done. 
		TxtReceived := ResponseBuilder.ToString; 
		ActualResponse.Clear();
		ActualResponse.AppendGeneric(ResponseBuilder.StringPointer,ResponseBuilder.Length); 
	END_IF

END_IF

_errorID := fb.nErrId;
END_METHOD

METHOD PRIVATE state_Sending : BOOL
VAR_INPUT
	RequestAdr		: POINTER TO BYTE; 
	RequestLength	: UDINT; 
END_VAR
VAR_IN_OUT
	ResponseBuilder		: FB_StringBuilder;
	Handle			: T_HSOCKET;
	CurrentState	: E_TcpState;		
END_VAR

VAR_INST
	DebugRequest	: BOOL; 
	fb				: FB_SocketSend; 
	ErrorID			: UDINT; 
	RequestTxt		: T_MAXSTRING;
	error			: T_MAXSTRING;
END_VAR


fb(
		sSrvNetId	:= _AmsNetId, 
		hSocket		:= Handle, 
		bExecute	:= NOT(_firstTimeInState),
		cbLen		:= RequestLength, 
		pSrc		:= RequestAdr, 
		tTimeout	:= T#500h, 
		bBusy		=> , 
		bError		=> , 
		nErrId		=> ErrorID);
		


IF fb.bError AND NOT(_firstTimeInState) THEN
	fb(bExecute := FALSE);
	error := ErrorIdToString(fb.nErrId); 
	CurrentState := E_TcpState.Disconnected;

ELSIF NOT(fb.bBusy) AND NOT(_firstTimeInState) THEN
	fb(bExecute := FALSE);
	ResponseBuilder.Clear(); // Clear response, ready for receiving new response.
	CurrentState := E_TcpState.Waiting;
END_IF


_errorID := fb.nErrId;
END_METHOD

METHOD PRIVATE state_Waiting : BOOL
VAR_INPUT
	WaitTime	: TIME; 
END_VAR
VAR_IN_OUT
	CurrentState	: E_TcpState;
END_VAR
VAR_INST
	TimesExecuted : UDINT; 
END_VAR
IF WaitTime < T#5MS THEN
	WaitTime := T#50MS;
END_IF

IF _timeInState >= WaitTime THEN
	TimesExecuted := TimesExecuted + 1; 
	CurrentState := E_TcpState.Receiving; 
END_IF
END_METHOD

METHOD PRIVATE UpdateMetrics : BOOL
VAR_IN_OUT
	CurrentState	: E_TcpState; 	


END_VAR

VAR_OUTPUT
	IdleTime	: TIME; 	
	TimeInState	: TIME; 
	CyclesInState : UDINT;
	FirstTimeInState	 : BOOL; 
	
END_VAR

VAR_INST
	_lastState	: E_TcpState; 
	_IdleTimer	: TON; 
	_StateTimer	: TON; 
	_ReceiveTimer : TON;
	
	_cycles		: UDINT;
END_VAR

_IdleTimer(		IN	:= CurrentState = E_TcpState.Connected,
				PT	:= T#200H,
				ET	=> IdleTime); 

_StateTimer(	IN	:= CurrentState = _lastState,
				PT	:= T#1000H,
				ET	=> TimeInState); 
				
_ReceiveTimer(	IN	:= CurrentState = E_TcpState.Receiving OR CurrentState = E_TcpState.Waiting,
				PT	:= T#2S,	// Timeout for Receiving data
				ET	=> ); 
				
				
IF CurrentState = _lastState THEN
	_cycles := _cycles + 1;
	FirstTimeInState := FALSE;
ELSE
	_cycles := 0; 
	FirstTimeInState := TRUE; 
END_IF

IF _ReceiveTimer.Q OR _IdleTimer.ET > T#5s THEN
	CurrentState := E_TcpState.Disconnecting;
END_IF
				
CyclesInState := _cycles; 		
				
				
				
				
				
_lastState := CurrentState;
END_METHOD

END_FUNCTION_BLOCK

// ---- MAIN.TcPOU
PROGRAM MAIN
VAR
	Data					: ST_DATA;
	
	
	// ============== Set input/output mode: 	StaticData, SimulinkPlant, VirtualPlant PhysicalPlant	
	EmulatedState 			: E_EmulatedState 		:= E_EmulatedState.VirtualPlant;		
	
END_VAR



//============ UPDATE DAQ =============	
P_UpdateDAQ(Data := Data);

//============ UPDATE HMI =============	
P_UpdateHmi(Data := Data);

END_PROGRAM

// ---- Main/Programs/P_UpdateHmi.TcPOU
PROGRAM P_UpdateHmi
VAR_IN_OUT
	Data		: ST_DATA;
END_VAR

Communication.ToHmi.Data	:= Data;

END_PROGRAM

// ---- DAQ/FromLib/Influxdb/Reader/FB_InfluxReader.TcPOU
FUNCTION_BLOCK FB_InfluxReader
VAR_INPUT
	Ip					: T_IPv4Addr := '127.0.0.1'; (* IP Adress for TCP/IP Server *)
	Port 				: UDINT := 8086; (* Port To Connect to *)
	ReplyReadInterval 	: TIME := T#200MS; (* Time for allowing server to start responding*)
	InfluxDatabase		: T_MAXSTRING;
	InfluxMeasurement	: T_MAXSTRING; 
	ValuesToFind		: DINT; 
	TimeOffset			: T_MAXSTRING; 
END_VAR
VAR_IN_OUT
		ValueNames			: ARRAY[0..50] OF T_MAXSTRING;
END_VAR
VAR_OUTPUT
		ValuesRead			: ARRAY[0..50] OF LREAL;
		CurrentState	: 	E_InfluxReaderState; 
		
END_VAR
VAR
	NamesLower 		: DINT;
	NamesUpper 		: DINT;
	NamesNumber		: DINT;
	iNames			: DINT; 
	iNamesAdded		: DINT; 
	                  
	ValuesLower		: DINT;
	ValuesUpper		: DINT;
	ValuesNumber	: DINT;
END_VAR

VAR
	iTest 	: UDINT; 
	ReadData		: BOOL; 
	
	
	LastState		: E_InfluxReaderState; 
	InStateCounter : TON; 
	
	tcp	: FB_TcpConnection;	
	
	http	: FB_StringBuilder; 
	query	: FB_StringBuilder; 
	
	QueryString	: STRING(500); 
	
	ResultsFound : UDINT;
END_VAR

// ========== Manage Stuff
	iTest := iTest + 1;
	
	tcp(	Ip 					:= Ip,//'192.168.1.209',
			Port				:= Port,
			ReplyReadInterval 	:= ReplyReadInterval); 
	
	InStateCounter(IN := CurrentState = LastState,
					PT := T#10S); 

// ========== Range calculations
	NamesLower 	 := 0;//LOWER_BOUND(ValueNames,1);
	NamesUpper 	 := 50;//UPPER_BOUND(ValueNames,1);
	NamesNumber	 := ABS(NamesUpper - NamesLower);
				 
	ValuesLower	 := 0;//LOWER_BOUND(ValuesRead,1);
	ValuesUpper	 := 50;//UPPER_BOUND(ValuesRead,1);
	ValuesNumber := ABS(ValuesUpper - ValuesLower);

// ========= Handle Timeout				
	IF InStateCounter.Q THEN	// Do To idle if no state change in 2min
		CurrentState := E_InfluxReaderState.Idle;
	END_IF

// ======== Read values				
	CASE CurrentState OF
		
		E_InfluxReaderState.Idle:
			IF ReadData THEN
				ReadData := FALSE;
				CurrentState	:= E_InfluxReaderState.Connecting;
			END_IF
	
		E_InfluxReaderState.Connecting:
			tcp.Connect();
			IF tcp.Connected THEN
				CurrentState	:= E_InfluxReaderState.Query;
			END_IF
		
		E_InfluxReaderState.Query:
			// eg: 'q=SELECT last(TestData),last(TestData1),last(TestData2) FROM test LIMIT 1'; 
			query.Clear(); 
			query.Append('q=SELECT ');
			iNamesAdded := 0; 
			FOR iNames := NamesLower TO NamesUpper DO
				query.Append('last(');
				query.Append(ValueNames[iNames]);
				query.Append(')');
				iNamesAdded := iNamesAdded + 1; 
				
				IF iNamesAdded = ValuesToFind THEN
					EXIT;
				ELSE
					query.Append(',');
				END_IF
			END_FOR
			
			query.Append(' FROM ');
			query.Append(InfluxMeasurement);
			
			IF len(TimeOffset) > 0 THEN
				query.Append(' WHERE time < now() - '); // JBM: Should it be WHERE time > now() - 10m?
				query.Append(TimeOffset);			
			END_IF
			
			
			query.AppendLine(' LIMIT 1');
		
			http.Clear(); 
			http.Append('POST /query?db=');
			http.Append(InfluxDatabase);  
			http.AppendLine(' HTTP/1.1');
			http.AppendLine('Host: BeckhoffIPC');
			http.AppendLine('User-Agent: TwinCAT HttpClient');
			http.AppendLine('Accept: */*');
			http.AppendLine('Content-Type: application/x-www-form-urlencoded');
			http.Append('Content-Length: ');
			http.AppendLine(TO_STRING(query.Length));
			http.AppendLine('');
			http.AppendGeneric(query.StringPointer,query.Length);	
				
			memcpy(ADR(QueryString), http.StringPointer, MIN(http.Length,SIZEOF(QueryString)));
			
			tcp.Send(http.StringPointer, http.Length);
			CurrentState	:= E_InfluxReaderState.ConvertingNumbers;
			

			
		E_InfluxReaderState.ConvertingNumbers:
		
			IF NOT(tcp.Busy) THEN
				QueryString := tcp.Response.ToString;
				ExtractNumbers(	InputString 	:= tcp.Response,
								ResultArray 	:= ValuesRead,
								NumbersToFind 	:= ValuesToFind,
								ValuesFound		=> ResultsFound); 
							
							CurrentState	:= E_InfluxReaderState.Disconnecting;
							tcp.Disconnect();
			END_IF
		
		
	
			
				
			
		E_InfluxReaderState.Disconnecting:				
			IF NOT(tcp.Connected) THEN
				CurrentState	:= E_InfluxReaderState.Idle;
			END_IF
	
	END_CASE

METHOD PRIVATE ExtractNumbers : BOOL
VAR_IN_OUT
	InputString : FB_StringBuilder; 
	ResultArray : ARRAY[0..50] OF LREAL; 
END_VAR


VAR_INPUT
	NumbersToFind	: DINT;	
END_VAR
VAR
	ActualNumbersToFind : DINT;
	iSearchNumber	: DINT;
END_VAR


VAR_OUTPUT
	
	ValuesFound : UDINT; 

END_VAR
VAR
	arLower	: DINT; 
	arUpper	: DINT; 
	
	iStartIndex : DINT; 
	
		searchString	: T_MAXSTRING := 'values';
		
	iNumberStart : DINT; 	
	iNumberEnd : DINT; 	
	iNumberLength : DINT; 
	
	numberTxt		: T_MAXSTRING;
	parsedNumber	: LREAL; 
END_VAR
VAR_INST
	Info	 : ARRAY[0..10] OF ST_NumberInString;
END_VAR
arLower := 0; 
arUpper := 50;

ActualNumbersToFind := MIN(NumbersToFind, arUpper - arLower); 

IF ActualNumbersToFind > 0 THEN

	iStartIndex := InputString.GetIndexOf('values',250);
	iStartIndex := InputString.GetIndexOf(',',TO_UDINT(iStartIndex)); // Position of first comma after Time info
	
	// EG: {"results":[{"statement_id":0,"series":[{"name":"test","columns":["time","last","last_1","last_2"],"values":[["1970-01-01T00:00:00Z",12344,12344.123123123,0.0123421342]]}]}]}$N
	
	iNumberEnd	 := iStartIndex;
	
	FOR iSearchNumber := 0 TO ActualNumbersToFind - 1 DO
		// Find each number
		iNumberStart := iNumberEnd +1;
		
		IF iSearchNumber < ActualNumbersToFind - 1 THEN
			iNumberEnd := InputString.GetIndexOf(',',TO_UDINT(iNumberStart+1));
		ELSE
			iNumberEnd := InputString.GetIndexOf(']',TO_UDINT(iNumberStart+1));
		END_IF
		
		iNumberLength := iNumberEnd - iNumberStart; 
		
		IF iNumberStart = -1 OR iNumberEnd = -1 THEN
			EXIT;
		END_IF
		
		// Copy txt to T_MAXSTRING
		numberTxt := ''; 
		
		memset(	destAddr	:= ADR(numberTxt),
				fillByte	:= 0,
				n			:= SIZEOF(T_MAXSTRING));
				
		memcpy(	destAddr 	:= ADR(numberTxt),
				srcAddr		:=  InputString.StringPointer+ TO_LWORD(iNumberStart), 
				n			:=  TO_UDINT(MIN(iNumberLength,SIZEOF(T_MAXSTRING))));
	
		parsedNumber := TO_LREAL(numberTxt);
		
		ResultArray[arLower + iSearchNumber] := parsedNumber; 
		
		IF iSearchNumber < 10 THEN
			info[iSearchNumber].StartIndex 	:= iNumberStart;
			info[iSearchNumber].EndIndex 	:= iNumberEnd;
			info[iSearchNumber].Length 		:= iNumberLength; 
			info[iSearchNumber].Txt 		:= numberTxt;
			info[iSearchNumber].Value 		:= parsedNumber; 
		END_IF
		
		
	END_FOR

	

END_IF
END_METHOD

METHOD ReadValues : BOOL
THIS^.ReadData := TRUE;
END_METHOD

END_FUNCTION_BLOCK

// ---- DAQ/InfluxReader/ExtractValuesFromInflux/fcnExtractInfluxData.TcPOU
FUNCTION fcnExtractInfluxData : BOOL
VAR_IN_OUT
	InputString : FB_StringBuilder; 
	ResultArray : ARRAY[*] OF LREAL; 
END_VAR


VAR_INPUT
	NumbersToFind	: DINT;	
END_VAR
VAR
	ActualNumbersToFind : DINT;
	iSearchNumber	: DINT;
END_VAR


VAR_OUTPUT
	
	ValuesFound : UDINT; 

END_VAR
VAR
	arLower	: DINT; 
	arUpper	: DINT; 
	
	iStartIndex : DINT; 
	
		searchString	: T_MAXSTRING := 'values';
		
	iNumberStart : DINT; 	
	iNumberEnd : DINT; 	
	iNumberLength : DINT; 
	
	numberTxt		: T_MAXSTRING;
	parsedNumber	: LREAL; 
	
	Info	 : ARRAY[0..10] OF ST_NumberInString;
END_VAR

arLower := LOWER_BOUND(ResultArray,1); 
arUpper := UPPER_BOUND(ResultArray,1); 

ActualNumbersToFind := MIN(NumbersToFind, arUpper - arLower); 

IF ActualNumbersToFind > 0 THEN

	iStartIndex := InputString.GetIndexOf('values',250);
	iStartIndex := InputString.GetIndexOf(',',iStartIndex); // Position of first comma after Time info
	
	// EG: {"results":[{"statement_id":0,"series":[{"name":"test","columns":["time","last","last_1","last_2"],"values":[["1970-01-01T00:00:00Z",12344,12344.123123123,0.0123421342]]}]}]}$N
	
	iNumberEnd	 := iStartIndex;
	
	FOR iSearchNumber := 0 TO ActualNumbersToFind - 1 DO
		// Find each number
		iNumberStart := iNumberEnd +1;
		
		IF iSearchNumber < ActualNumbersToFind - 1 THEN
			iNumberEnd := InputString.GetIndexOf(',',iNumberStart+1);
		ELSE
			iNumberEnd := InputString.GetIndexOf(']',iNumberStart+1);
		END_IF
		
		iNumberLength := iNumberEnd - iNumberStart; 
		
		// Copy txt to T_MAXSTRING
		numberTxt := ''; 
		
		memset(	destAddr	:= ADR(numberTxt),
				fillByte	:= 0,
				n			:= SIZEOF(T_MAXSTRING));
				
		memcpy(	destAddr 	:= ADR(numberTxt),
				srcAddr		:=  InputString.StringPointer+ TO_LWORD(iNumberStart), 
				n			:=  TO_UDINT(MIN(iNumberLength,SIZEOF(T_MAXSTRING))));
	
		parsedNumber := TO_LREAL(numberTxt);
		
		ResultArray[arLower + iSearchNumber] := parsedNumber; 
		
		IF iSearchNumber < 10 THEN
			info[iSearchNumber].StartIndex 	:= iNumberStart;
			info[iSearchNumber].EndIndex 	:= iNumberEnd;
			info[iSearchNumber].Length 		:= iNumberLength; 
			info[iSearchNumber].Txt 		:= numberTxt;
			info[iSearchNumber].Value 		:= parsedNumber; 
		END_IF
		
		
	END_FOR

	

END_IF

END_FUNCTION

// ---- DAQ/InfluxReader/FB_Flender_DamageReader.TcPOU
FUNCTION_BLOCK FB_Flender_DamageReader
VAR_INPUT
	TimeOffset 		: T_MAXSTRING; 
	ReadInterval 	: TIME := T#1M; 
	Ip				: T_IPv4Addr := '127.0.0.1'; 
	
END_VAR
VAR
	iTest 	: UDINT; 
	
	Timer : TON; 
	bRead : BOOL; 
	
	Tags 	: ARRAY[0..50] OF T_MAXSTRING;
	Values 	: ARRAY[0..50] OF LREAL; 
	
	reader	: FB_InfluxReader; 
	CurrentState : 	E_InfluxReaderState;
END_VAR
VAR_IN_OUT
	Dmg_Foundation 	: LREAL;
	Dmg_Footplates 	: LREAL;
	Dmg_MBS			: LREAL;	
	Dmg_LU1			: LREAL; 
	Dmg_LU2			: LREAL; 
END_VAR

iTest := iTest + 1;

Timer( 	IN 	:= NOT(Timer.Q),
		PT 	:= ReadInterval,
		Q	=> bRead); 

IF bRead THEN
	bRead := FALSE;
	reader.ReadValues();
END_IF
// ========= Setup Values
	Tags[0] := 'General_Foundation_Lu1';
	Tags[1] := 'General_Foundation_Lu2';
	
	Tags[2] := 'General_Footplates_Lu1';
	Tags[3] := 'General_Footplates_Lu2';
	
	Tags[4] := 'General_MBS_Lu1';
	Tags[5] := 'General_MBS_Lu2';
	
	Tags[6] := 'General_Platform_Lu1';
	Tags[7] := 'General_Platform_Lu2';

// ======== Run Reader
	reader(	Ip					:= Ip, 
			Port				:= 8086, 
			ReplyReadInterval	:= T#200MS, 
			InfluxDatabase		:= 'RD_Damage', 
			InfluxMeasurement	:= 'DamageCalculation', 
			ValuesToFind		:= 8, 
			ValueNames			:= Tags,
			TimeOffset			:= TimeOffset,
			ValuesRead			=> Values,
			CurrentState		=> CurrentState);
		
		
// ======= Output Values
	Dmg_Foundation 	:= UpdateCurrentValue(Dmg_Foundation, Values[0], Values[1]);
	Dmg_Footplates 	:= UpdateCurrentValue(Dmg_Footplates, Values[2], Values[3]);
	Dmg_MBS			:= UpdateCurrentValue(Dmg_MBS, Values[4], Values[5]); 
	Dmg_LU1			:= UpdateCurrentValue(Dmg_LU1, Values[6], 0);
	Dmg_LU2			:= UpdateCurrentValue(Dmg_LU1, Values[7], 0);

METHOD PRIVATE UpdateCurrentValue : LREAL
VAR_INPUT
	CurrentValue : LREAL;
	Lu1Value	: LREAL;
	Lu2Value 	: LREAL; 
END_VAR
VAR
	newestMaxValue : LREAL; 
	outputValue : LREAL;
END_VAR


newestMaxValue := MAX(Lu1Value, Lu2Value);


outputValue := MAX(CurrentValue, newestMaxValue); 

UpdateCurrentValue := outputValue;
END_METHOD

END_FUNCTION_BLOCK

// ---- DAQ/InfluxReader/P_FlenderGetDamage.TcPOU
PROGRAM P_FlenderGetDamage
VAR_IN_OUT
	DmgValue 	: ST_DamageCounter;	
END_VAR
VAR
	
	Dmg		 	: FB_Flender_DamageReader;
	Dmg1h		: FB_Flender_DamageReader;
	Dmg24h		: FB_Flender_DamageReader;

END_VAR
VAR
	InfluxIp				: T_IPv4Addr := '10.10.0.122'; 
	ReadInterval 			: TIME := T#1M; 
	
END_VAR
VAR PERSISTENT
	Dmg_Foundation_Current 	: LREAL;
    Dmg_Footplates_Current 	: LREAL;
    Dmg_MBS_Current			: LREAL;
    Dmg_Lu1_Current			: LREAL;
	Dmg_Lu2_Current			: LREAL;
	
	Dmg_Foundation_1h 		: LREAL;
    Dmg_Footplates_1h 		: LREAL;
    Dmg_MBS_1h				: LREAL;
    Dmg_Lu1_1h				: LREAL;
 	Dmg_Lu2_1h				: LREAL;
	                    	
	Dmg_Foundation_24h 		: LREAL;
    Dmg_Footplates_24h 		: LREAL;
    Dmg_MBS_24h				: LREAL;
    Dmg_Lu1_24h				: LREAL;
	Dmg_Lu2_24h				: LREAL;

END_VAR

// ============= Get Data
	Dmg(
		TimeOffset		:= '', 
		ReadInterval	:= ReadInterval, 
		Ip				:= InfluxIp, 
		Dmg_Foundation	:= Dmg_Foundation_Current, 
		Dmg_Footplates	:= Dmg_Footplates_Current, 
		Dmg_MBS			:= Dmg_MBS_Current, 
		Dmg_Lu1			:= Dmg_Lu1_Current,
		Dmg_Lu2			:= Dmg_Lu2_Current	);
	
	Dmg1h(
		TimeOffset		:= '1h', 
		ReadInterval	:= ReadInterval, 
		Ip				:= InfluxIp, 
		Dmg_Foundation	:= Dmg_Foundation_1h, 
		Dmg_Footplates	:= Dmg_Footplates_1h, 
		Dmg_MBS			:= Dmg_MBS_1h, 
		Dmg_Lu1			:= Dmg_Lu1_1h,
		Dmg_Lu2			:= Dmg_Lu2_1h	);
		
	Dmg24h(
		TimeOffset		:= '24h', 
		ReadInterval	:= ReadInterval, 
		Ip				:= InfluxIp, 
		Dmg_Foundation	:= Dmg_Foundation_24h, 
		Dmg_Footplates	:= Dmg_Footplates_24h, 
		Dmg_MBS			:= Dmg_MBS_24h, 
		Dmg_Lu1			:= Dmg_Lu1_24h,
		Dmg_Lu2			:= Dmg_Lu2_24h	);
		
		
// ============= Calculate Display Values

DmgValue.FootPlatesDmg.AccumulatedDmg.fValue 	:= Dmg_Footplates_Current;
DmgValue.FootPlatesDmg.DmgRate1hr.fValue 		:= Dmg_Footplates_Current - Dmg_Footplates_1h;
DmgValue.FootPlatesDmg.DmgRate1day.fValue 		:= Dmg_Footplates_Current - Dmg_Footplates_24h; 

DmgValue.FoundationDmg.AccumulatedDmg.fValue 	:= Dmg_Foundation_Current;
DmgValue.FoundationDmg.DmgRate1hr.fValue 		:= Dmg_Foundation_Current - Dmg_Foundation_1h;
DmgValue.FoundationDmg.DmgRate1day.fValue 		:= Dmg_Foundation_Current - Dmg_Foundation_24h; 

DmgValue.Lu1Dmg.AccumulatedDmg.fValue 			:= Dmg_Lu1_Current;
DmgValue.Lu1Dmg.DmgRate1hr.fValue 				:= Dmg_Lu1_Current - Dmg_Lu1_1h;
DmgValue.Lu1Dmg.DmgRate1day.fValue 				:= Dmg_Lu1_Current - Dmg_Lu1_24h; 

DmgValue.Lu2Dmg.AccumulatedDmg.fValue 			:= Dmg_Lu2_Current;
DmgValue.Lu2Dmg.DmgRate1hr.fValue 				:= Dmg_Lu2_Current - Dmg_Lu2_1h;
DmgValue.Lu2Dmg.DmgRate1day.fValue 				:= Dmg_Lu2_Current - Dmg_Lu2_24h; 

DmgValue.MbsDmg.AccumulatedDmg.fValue 			:= Dmg_MBS_Current;
DmgValue.MbsDmg.DmgRate1hr.fValue 				:= Dmg_MBS_Current - Dmg_MBS_1h;
DmgValue.MbsDmg.DmgRate1day.fValue 				:= Dmg_MBS_Current - Dmg_MBS_24h;

END_PROGRAM
